(* CODESYS project CfUnit.project
   Project Profile: MachineProfile

Project tree, tasks and I/O mapping:
  Device : XP325, Altus S.A., order no. XP325, version 1.0.0.48
    application Application
      libraries: NextoStandard, 1.1.0.26 (WAA); LibIntegratedIo, 1.0.0.11 (Manufacturer); LibDataTypes, 1.0.0.0 (Manufacturer); XP325 Diagnostic Structs, 1.0.0.9 (Manufacturer); Standard, 3.5.12.0 (System)
      task MainTask (cyclic, interval 20 ms, priority 13, watchdog 1000 ms x 1) calls MainPrg
      SystemGVLs/
        global variables System_Diagnostics
        global variables IntegratedIO
      UserGVLs/
        global variables Qualities
        global variables ReqDiagnostics
        global variables Disables
      SystemPOUs/
        program MainPrg [ST]
      UserPOUs/
        program UserPrg [LD]
        program StartPrg [LD]
    Configuration : XP, WAA, order no. Configuration, version 1.1.1.2
        settings: Machine Profile = TRUE
      XP325 : XP325, Altus S.A., order no. XP325, version 1.0.0.48
          settings: DC sync0 cycletime = 5000; IOModule's Address for interrupt = 255; Complete Access = TRUE; CurrentProjectProfileParameter = 'MachineProfile'
        <Vazio>
        COM 1
        NET 1
        CAN
        Integrated I/O
*)

// Device/Application/SystemGVLs/System_Diagnostics
VAR_GLOBAL
	//DG_XP325 diagnostics variable
	DG_XP325 : T_DIAG_XP325_1;
END_VAR

// Device/Application/UserGVLs/Qualities
VAR_GLOBAL
END_VAR

// Device/Application/UserGVLs/ReqDiagnostics
VAR_GLOBAL
END_VAR

// Device/Application/UserGVLs/Disables
VAR_GLOBAL
END_VAR

// Device/Application/SystemGVLs/IntegratedIO
VAR_GLOBAL

	// Structured tags for I/O points
	DigitalInputs  : T_DIGITAL_INPUTS_1;                                 // Digital Inputs structure
	DigitalOutputs : T_DIGITAL_OUTPUTS_1;                                // Digital Outputs structure
	FastInputs     : T_FAST_INPUTS_1;                                    // Fast Inputs structure
	FastOutputs    : T_FAST_OUTPUTS_1;                                   // Fast Outputs structure
	AnalogInputs   : T_ANALOG_INPUTS_1;                                  // Analog Inputs structure
	AnalogOutputs  : T_ANALOG_OUTPUTS_1;                                 // Analog Ouputs structure
	RtdInputs      : T_RTD_INPUTS_1;                                     // RTD Inputs structure

	// Direct tags for I/O points
	I0             : REFERENCE TO BYTE   := DigitalInputs.Group0.Value;  // Digital Inputs Group 0
	I1             : REFERENCE TO BYTE   := DigitalInputs.Group1.Value;  // Digital Inputs Group 1

	Q0             : REFERENCE TO BYTE   := DigitalOutputs.Group0.Value; // Digital Outputs Group 0
	Q1             : REFERENCE TO BYTE   := DigitalOutputs.Group1.Value; // Digital Outputs Group 1

	AI0            : REFERENCE TO INT    := AnalogInputs.AI0;            // Analog Input 0
	AI1            : REFERENCE TO INT    := AnalogInputs.AI1;            // Analog Input 1
	AI2            : REFERENCE TO INT    := AnalogInputs.AI2;            // Analog Input 2
	AI3            : REFERENCE TO INT    := AnalogInputs.AI3;            // Analog Input 3
	AI4            : REFERENCE TO INT    := AnalogInputs.AI4;            // Analog Input 4

	AO0            : REFERENCE TO INT    := AnalogOutputs.AO0;           // Analog Output 0
	AO1            : REFERENCE TO INT    := AnalogOutputs.AO1;           // Analog Output 1
	AO2            : REFERENCE TO INT    := AnalogOutputs.AO2;           // Analog Output 2
	AO3            : REFERENCE TO INT    := AnalogOutputs.AO3;           // Analog Output 3

	RI0            : REFERENCE TO INT    := RtdInputs.R00;               // RTD Input 0
	RI1            : REFERENCE TO INT    := RtdInputs.R01;               // RTD Input 1

END_VAR

// Device/Application/SystemPOUs/MainPrg
(*Main POU associated with MainTask that calls StartPrg, UserPrg/ActivePrg and NonSkippedPrg. This POU is blocked to edit.*)
PROGRAM MainPrg
VAR
   isFirstCycle : BOOL := TRUE;
END_VAR

IF isFirstCycle THEN
   StartPrg();
   isFirstCycle := FALSE;
ELSE
   UserPrg();
END_IF;

END_PROGRAM

// Device/Application/UserPOUs/StartPrg
(*The code inserted by the user into this POU is executed once after startup. Before this fist cycle it is not executed again. In case of redundant system, this one is executed in both CPUs during the startup.*)
PROGRAM StartPrg
VAR
END_VAR

// NETWORK 1

END_PROGRAM

// Device/Application/UserPOUs/UserPrg
(*The main code inserted by the user and executed associated with the MainTask must be inserted into this POU.*)
PROGRAM UserPrg
VAR
END_VAR

// NETWORK 1

END_PROGRAM
